FUNCTION_BLOCK FB_ErrorHandling
VAR_INPUT
	xEStop: BOOL;
END_VAR
VAR_OUTPUT
	eErrorHandling: E_ErrorHandling;
END_VAR
VAR
END_VAR

IF xEStop THEN
	eErrorHandling:= Emergency;
ELSIF IOs.xMC_HasError THEN
		eErrorHandling:= Fault;
		ELSE
			eErrorHandling:= No_Error;
END_IF

END_FUNCTION_BLOCK

(* stored: Version 1.1.0.1
   POU FB_ErrorHandling: Id {fc95b0d0-6a29-4392-a6b9-d4bc4d625903}, SpecialFunc None *)
